PROGRAM MAIN
VAR
	Hethong : FB_System;
END_VAR

Hethong();

END_PROGRAM

(* stored: Version 1.1.0.1, ProductVersion 3.1.4024.16
   POU MAIN: Id {487ac2db-d967-499e-ac9e-fd5c6a60eb36}, SpecialFunc None *)
